Universal Robots PolyScope program: ejercicio_1.urp

Program ejercicio_1 (installation=ejercicio_1 directory=/home/ur/ursim-current/programs/Entregables/Easy programing/ejercicio 1 createdIn=5.9.4.1031232 lastSavedIn=5.9.4.1031232 robotSerialNumber=20195599999)
Calibrated DH parameters: a=[0, -0.425, -0.3922, 0, 0, 0]; d=[0.1625, 0, 0, 0.1333, 0.0997, 0.0996]; alpha=[1.570796, 0, 0, 1.570796, -1.570796, 0]; deltaTheta=[0, 0, 0, 0, 0, 0]
Robot Program (runOnlyOnce=false)
  Folder variables
    pi := 3.1416
    pick_arriba := p[0.5,0,0.25,0,pi,0]
    pick_abajo := p[0.5,0,0,0,pi,0]
    place_arriba := p[0.5,0.25,0.25,0,pi,0]
    place_abajo := p[0.5,0.25,0,0,pi,0]
    safe_point := [0,-pi/4,-pi/2,-3*pi/4,pi/2,0]
  Popup Message (haltProgram=false message=El programa va a comenzar inputType=Text)
  MoveJ speed 60 deg/s, acceleration 80 deg/s^2 (useActiveTCP=false) tcp=TCP_1; feature=Base
    Waypoint Waypoint (Variable): variable=safe_point
  MoveJ speed 60 deg/s, acceleration 80 deg/s^2 (useActiveTCP=false) tcp=TCP_1; feature=Base
    Waypoint Waypoint (Variable): variable=pick_arriba
  MoveL speed 250 mm/s, acceleration 1200 mm/s^2 (useActiveTCP=false) tcp=TCP_1; feature=Base
    Waypoint Waypoint (Variable): variable=pick_abajo
  'PICK'
  Wait Sleep waitTime=1
  MoveL speed 250 mm/s, acceleration 1200 mm/s^2 (useActiveTCP=false) tcp=TCP_1; feature=Base
    Waypoint Waypoint (Variable): variable=pick_arriba
  MoveJ speed 60 deg/s, acceleration 80 deg/s^2 (useActiveTCP=false) tcp=TCP_1; feature=Base
    Waypoint Waypoint (Variable): variable=place_arriba
  MoveL speed 250 mm/s, acceleration 1200 mm/s^2 (useActiveTCP=false) tcp=TCP_1; feature=Base
    Waypoint Waypoint (Variable): variable=place_abajo
  'PLACE'
  Wait Sleep waitTime=1
  MoveL speed 250 mm/s, acceleration 1200 mm/s^2 (useActiveTCP=false) tcp=TCP_1; feature=Base
    Waypoint Waypoint (Variable): variable=place_arriba
  MoveJ speed 60 deg/s, acceleration 80 deg/s^2 (useActiveTCP=false) tcp=TCP_1; feature=Base
    Waypoint Waypoint (Variable): variable=safe_point
  Popup Message (haltProgram=true message=El programa ha acabado inputType=Text)
